// TIA Portal V21 export
FUNCTION "AoFc" : Void   // FC106, LAD
{ S7_Optimized_Access := 'TRUE' }
// stored: AutoNumber false, SetENOAutomatically false
   VAR_TEMP   // added for the SCL form of the ladder/FBD networks
      _w1 : Bool;
      _w2 : Bool;
   END_VAR
BEGIN

REGION Network 1: "AoDb"
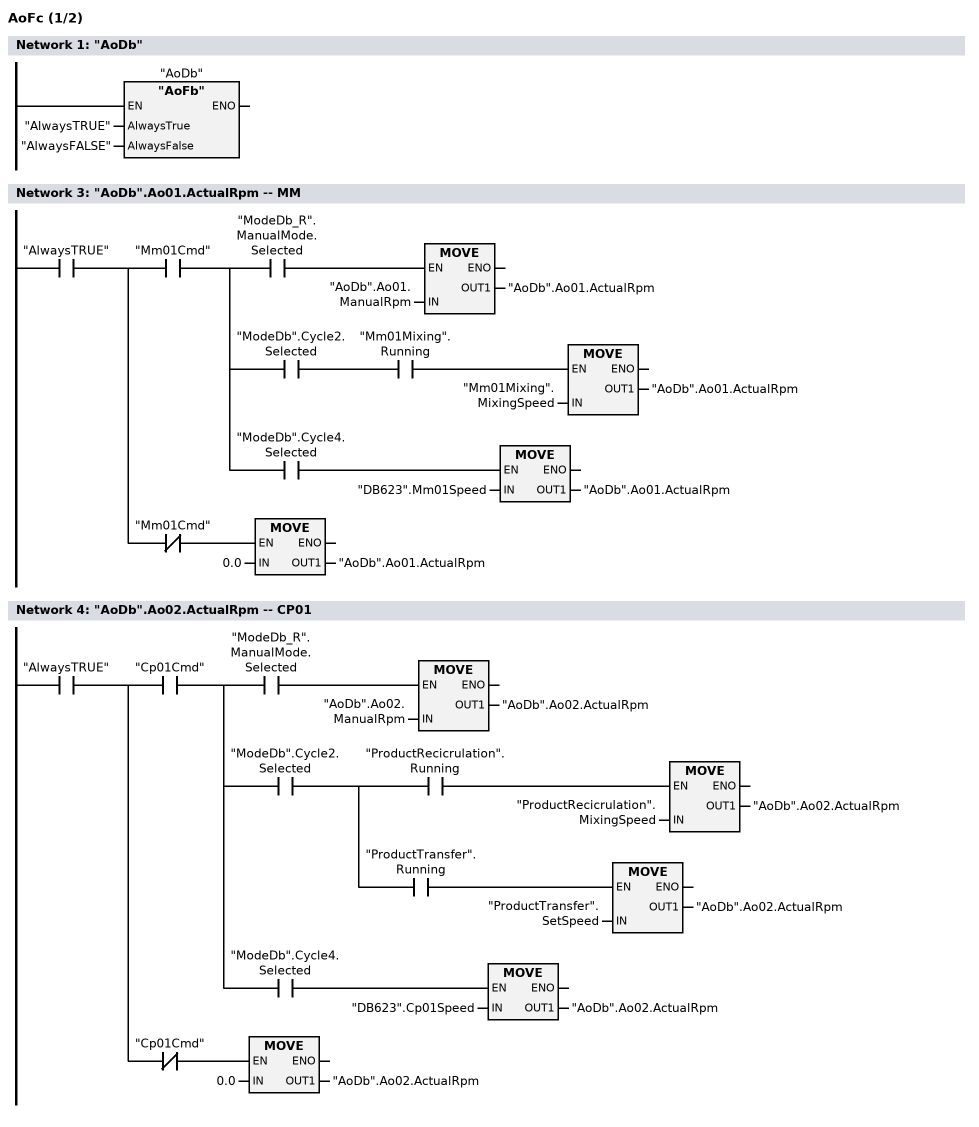
   RUNG wire#powerrail
      "AoDb"(AlwaysTrue := "AlwaysTRUE", AlwaysFalse := "AlwaysFALSE")
   END_RUNG
   // the same network as SCL:
   "AoDb"(AlwaysTrue := "AlwaysTRUE", AlwaysFalse := "AlwaysFALSE");   // "AoFb"
END_REGION

REGION Network 2 (SCL): Output to PLC Tag
   "Mm01Ref" := "AoDb".Ao01.Output;
   "Cp01Ref" := "AoDb".Ao02.Output;
   "Cv01"    :=  "AoDb".Ao03.Output;
   "AoSpare1" := "AoDb".Ao04.Output;
   "AoSpare2" := "AoDb".Ao05.Output;
   "AoSpare3" := "AoDb".Ao06.Output;
   "AoSpare4" := "AoDb".Ao07.Output;
   "AoSpare5" := "AoDb".Ao08.Output;
END_REGION

REGION Network 3: "AoDb".Ao01.ActualRpm -- MM
   RUNG wire#powerrail
      Contact( "AlwaysTRUE" )
      wire#w1
      Contact( "Mm01Cmd" )
      wire#w2
      Contact( "ModeDb_R".ManualMode.Selected )
      Move(in := "AoDb".Ao01.ManualRpm, out1 => "AoDb".Ao01.ActualRpm)
   END_RUNG
   RUNG wire#w2
      Contact( "ModeDb".Cycle2.Selected )
      Contact( "Mm01Mixing".Running )
      Move(in := "Mm01Mixing".MixingSpeed, out1 => "AoDb".Ao01.ActualRpm)
   END_RUNG
   RUNG wire#w2
      Contact( "ModeDb".Cycle4.Selected )
      Move(in := "DB623".Mm01Speed, out1 => "AoDb".Ao01.ActualRpm)
   END_RUNG
   RUNG wire#w1
      I_Contact( "Mm01Cmd" )
      Move(in := 0.0, out1 => "AoDb".Ao01.ActualRpm)
   END_RUNG
   // the same network as SCL:
   #_w1 := "AlwaysTRUE" AND "Mm01Cmd";
   IF #_w1 AND "ModeDb_R".ManualMode.Selected THEN "AoDb".Ao01.ActualRpm := "AoDb".Ao01.ManualRpm; END_IF;
   IF #_w1 AND "ModeDb".Cycle2.Selected AND "Mm01Mixing".Running THEN
       "AoDb".Ao01.ActualRpm := "Mm01Mixing".MixingSpeed;
   END_IF;
   IF #_w1 AND "ModeDb".Cycle4.Selected THEN "AoDb".Ao01.ActualRpm := "DB623".Mm01Speed; END_IF;
   IF "AlwaysTRUE" AND NOT "Mm01Cmd" THEN "AoDb".Ao01.ActualRpm := 0.0; END_IF;
END_REGION

REGION Network 4: "AoDb".Ao02.ActualRpm -- CP01
   RUNG wire#powerrail
      Contact( "AlwaysTRUE" )
      wire#w1
      Contact( "Cp01Cmd" )
      wire#w2
      Contact( "ModeDb_R".ManualMode.Selected )
      Move(in := "AoDb".Ao02.ManualRpm, out1 => "AoDb".Ao02.ActualRpm)
   END_RUNG
   RUNG wire#w2
      Contact( "ModeDb".Cycle2.Selected )
      wire#w3
      Contact( "ProductRecicrulation".Running )
      Move(in := "ProductRecicrulation".MixingSpeed, out1 => "AoDb".Ao02.ActualRpm)
   END_RUNG
   RUNG wire#w3
      Contact( "ProductTransfer".Running )
      Move(in := "ProductTransfer".SetSpeed, out1 => "AoDb".Ao02.ActualRpm)
   END_RUNG
   RUNG wire#w2
      Contact( "ModeDb".Cycle4.Selected )
      Move(in := "DB623".Cp01Speed, out1 => "AoDb".Ao02.ActualRpm)
   END_RUNG
   RUNG wire#w1
      I_Contact( "Cp01Cmd" )
      Move(in := 0.0, out1 => "AoDb".Ao02.ActualRpm)
   END_RUNG
   // the same network as SCL:
   #_w1 := "AlwaysTRUE" AND "Cp01Cmd";
   IF #_w1 AND "ModeDb_R".ManualMode.Selected THEN "AoDb".Ao02.ActualRpm := "AoDb".Ao02.ManualRpm; END_IF;
   #_w2 := #_w1 AND "ModeDb".Cycle2.Selected;
   IF #_w2 AND "ProductRecicrulation".Running THEN
       "AoDb".Ao02.ActualRpm := "ProductRecicrulation".MixingSpeed;
   END_IF;
   IF #_w2 AND "ProductTransfer".Running THEN "AoDb".Ao02.ActualRpm := "ProductTransfer".SetSpeed; END_IF;
   IF #_w1 AND "ModeDb".Cycle4.Selected THEN "AoDb".Ao02.ActualRpm := "DB623".Cp01Speed; END_IF;
   IF "AlwaysTRUE" AND NOT "Cp01Cmd" THEN "AoDb".Ao02.ActualRpm := 0.0; END_IF;
END_REGION

REGION Network 5: CV01
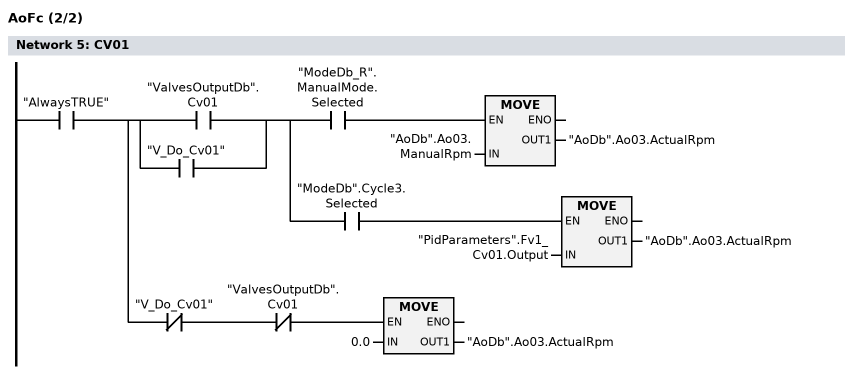
   RUNG wire#powerrail
      Contact( "AlwaysTRUE" )
      wire#w1
      Contact( "ValvesOutputDb".Cv01 )
      wire#w2
      Contact( "ModeDb_R".ManualMode.Selected )
      Move(in := "AoDb".Ao03.ManualRpm, out1 => "AoDb".Ao03.ActualRpm)
   END_RUNG
   RUNG wire#w1
      Contact( "V_Do_Cv01" )
   END_RUNG wire#w2
   RUNG wire#w2
      Contact( "ModeDb".Cycle3.Selected )
      Move(in := "PidParameters".Fv1_Cv01.Output, out1 => "AoDb".Ao03.ActualRpm)
   END_RUNG
   RUNG wire#w1
      I_Contact( "V_Do_Cv01" )
      I_Contact( "ValvesOutputDb".Cv01 )
      Move(in := 0.0, out1 => "AoDb".Ao03.ActualRpm)
   END_RUNG
   // the same network as SCL:
   #_w1 := "AlwaysTRUE" AND ("ValvesOutputDb".Cv01 OR "V_Do_Cv01");
   IF #_w1 AND "ModeDb_R".ManualMode.Selected THEN "AoDb".Ao03.ActualRpm := "AoDb".Ao03.ManualRpm; END_IF;
   IF #_w1 AND "ModeDb".Cycle3.Selected THEN
       "AoDb".Ao03.ActualRpm := "PidParameters".Fv1_Cv01.Output;
   END_IF;
   IF "AlwaysTRUE" AND NOT "V_Do_Cv01" AND NOT "ValvesOutputDb".Cv01 THEN
       "AoDb".Ao03.ActualRpm := 0.0;
   END_IF;
END_REGION
END_FUNCTION
